(* IEC 61131-3 sources: beckhoffAutomationInterface/ST/Shark/App/Shark/Config/Machine, 12 files *)

(* ---- GVL_ChuckVacuumSystem.st ---- *)
(* CONFIG_TIER: 1-MACHINE  -- Update all values for every new machine build. *)
(* Chuck vacuum zone size thresholds for the Shark system.
   Maps wafer diameter [mm] to vacuum zone selection:
     diameter <= CHUCK_ZONE_SMALL_MAX  -> zone 1 (small)
     diameter <= CHUCK_ZONE_MEDIUM_MAX -> zone 2 (medium)
     diameter >  CHUCK_ZONE_MEDIUM_MAX -> zone 3 (large) *)
{attribute 'qualified_only'}
VAR_GLOBAL CONSTANT
    CHUCK_ZONE_SMALL_MAX  : INT := 150;   // [mm] upper bound for small-wafer zone
    CHUCK_ZONE_MEDIUM_MAX : INT := 200;   // [mm] upper bound for medium-wafer zone
END_VAR

(* ---- GVL_DIOConfig.st ---- *)
(* CONFIG_TIER: 1-MACHINE  -- Update all values for every new machine build. *)
(* Digital I/O channel counts for the Shark system.
   Values must match the extent of the corresponding E_*Identifier enums.
   Absorbs the old GVL_DigitalInputSystem and GVL_DigitalOutputSystem files. *)
{attribute 'qualified_only'}
VAR_GLOBAL CONSTANT
    // Digital I/O channel counts (must match the extent of their E_*Identifier enums)
    DI_COUNT : INT := 12;   // E_DigitalInputIdentifier  (was GVL_DigitalInputSystem.INPUT_COUNT)
    DO_COUNT : INT := 16;   // E_DigitalOutputIdentifier (was GVL_DigitalOutputSystem.OUTPUT_COUNT)

    // Outputs activated once on first boot (section 8 one-time init)
    // To add a new auto-start output: increment AUTO_START_DO_COUNT and add the identifier.
    AUTO_START_DO_COUNT   : INT := 3;
    AUTO_START_DO_OUTPUTS : ARRAY[1..3] OF INT := [
        E_DigitalOutputIdentifier.LGHT_CMR_TOP,    // Top camera light
        E_DigitalOutputIdentifier.LGHT_CMR_SIDE,   // Side camera light
        E_DigitalOutputIdentifier.CHIL_PWR         // Chiller power
    ];
END_VAR

(* ---- GVL_DoorSystem.st ---- *)
(* CONFIG_TIER: 1-MACHINE  -- Update all values for every new machine build. *)
(* Door subsystem sizing constants for the Shark system.
   DOOR_SENSOR_COUNT must match the number of proximity sensors wired
   to E_DigitalInputIdentifier door entries.
   DOOR_LOCK_COUNT must match the number of electromechanical locks
   wired to E_DigitalOutputIdentifier lock entries (FL, FR). *)
{attribute 'qualified_only'}
VAR_GLOBAL CONSTANT
    DOOR_SENSOR_COUNT : INT := 9;   // Proximity sensors total
    DOOR_LOCK_COUNT   : INT := 2;   // Electromechanical locks (FL, FR)
END_VAR

(* ---- GVL_FlowSystem.st ---- *)
(* CONFIG_TIER: 1-MACHINE  -- Update all values for every new machine build. *)
{attribute 'qualified_only'}
VAR_GLOBAL CONSTANT
    // Flow Ranges - Precursor MFC (0-25 sccm)
    MIN_FLOW_PRECURSOR_SCCM : REAL := 0.0;
    MAX_FLOW_PRECURSOR_SCCM : REAL := 25.0;

    // Flow Ranges - Reactant MFC (0-25 sccm)
    MIN_FLOW_REACTANT_SCCM  : REAL := 0.0;
    MAX_FLOW_REACTANT_SCCM  : REAL := 25.0;

    // Flow Ranges - Inert MFC (0-500 sccm)
    MIN_FLOW_INERT_SCCM     : REAL := 0.0;
    MAX_FLOW_INERT_SCCM     : REAL := 500.0;

    // System Configuration
    FLOW_ZONE_COUNT          : INT := 3;

    // Tolerance for setpoint boundary detection
    SETPOINT_TOLERANCE       : REAL := 0.01;
END_VAR

(* ---- GVL_HumiditySystem.st ---- *)
(* CONFIG_TIER: 1-MACHINE  -- Update all values for every new machine build.
   Scaling for the MDP5001_300_7E2119CA humidity channel on the Shark TH sensor pair.
   Humidity channel uses standard 0-30518 full-scale.
   Temperature channel has moved to GVL_TemperatureSystem (AMBT_TEMP_*). *)
{attribute 'qualified_only'}
VAR_GLOBAL CONSTANT
    // AMBT_HUMID: Ambient relative humidity [%RH]
    AMBT_HUMID_RAW_MIN    : LREAL := 0.0;
    AMBT_HUMID_RAW_MAX    : LREAL := 30518.0;
    AMBT_HUMID_SCALED_MIN : LREAL := 0.0;    // %RH
    AMBT_HUMID_SCALED_MAX : LREAL := 100.0;  // %RH

END_VAR

(* ---- GVL_PressureSystem.st ---- *)
(* CONFIG_TIER: 1-MACHINE  -- Update all values for every new machine build. *)
{attribute 'qualified_only'}
VAR_GLOBAL CONSTANT
    // Pressure Sensor Count (analog read-only sensors)
    SENSOR_COUNT     : INT := 4;

    // Pressure Controller Count (Bronkhorst Modbus, managed by PRG_BronkhorstPressure)
    CONTROLLER_COUNT : INT := 2;

    // Pressure Limits
    MIN_PRESSURE_BAR : REAL := 0.0;
    MAX_PRESSURE_BAR : REAL := 3.0;

    // Pressure Controller Constants (Bronkhorst Modbus needle valves)
    MIN_PRESSURE_CTRL_BAR  : REAL := 0.0;
    MAX_PRESSURE_CTRL_BAR  : REAL := 3.0;
    SETPOINT_TOLERANCE     : REAL := 0.01;
    MODBUS_FIRST_SLAVE_ADDRESS : BYTE := 1;

    // Sensor-specific raw scaling (from old FB_PressureSensorManager)
    // PSNS_A_DST: 0-30518 raw → 0.0-3.0 bar(a)
    PSNS_A_DST_RAW_MIN      : LREAL := 0.0;
    PSNS_A_DST_RAW_MAX      : LREAL := 30518.0;
    PSNS_A_DST_SCALED_MIN   : LREAL := 0.0;
    PSNS_A_DST_SCALED_MAX   : LREAL := 3.0;

    // PSNS_B_DST: 0-30518 raw → 0.0-3.0 bar(a)
    PSNS_B_DST_RAW_MIN      : LREAL := 0.0;
    PSNS_B_DST_RAW_MAX      : LREAL := 30518.0;
    PSNS_B_DST_SCALED_MIN   : LREAL := 0.0;
    PSNS_B_DST_SCALED_MAX   : LREAL := 3.0;

    // PSNS_AB_EXH: 0-30518 raw → 0.0-1.0 bar(a)
    PSNS_AB_EXH_RAW_MIN     : LREAL := 0.0;
    PSNS_AB_EXH_RAW_MAX     : LREAL := 30518.0;
    PSNS_AB_EXH_SCALED_MIN  : LREAL := 0.0;
    PSNS_AB_EXH_SCALED_MAX  : LREAL := 1.0;

    // PSNS_CHK_VAC: 3052-15259 raw → 1.01325-0.00325 bar(a) [INVERTED]
    // NOTE: Physical relationship is inverted — higher raw = lower pressure (more vacuum).
    //       FB_AnalogSensor requires ascending ranges, so we store ascending params here.
    //       Reading will be physically inverted: actual_bar = 1.0165 - sensor_reading
    PSNS_CHK_VAC_RAW_MIN    : LREAL := 3052.0;
    PSNS_CHK_VAC_RAW_MAX    : LREAL := 15259.0;
    PSNS_CHK_VAC_SCALED_MIN : LREAL := 0.00325;
    PSNS_CHK_VAC_SCALED_MAX : LREAL := 1.01325;
END_VAR

(* ---- GVL_Spectrometer.st ---- *)
(* CONFIG_TIER: 1-MACHINE  -- Update all values for every new machine build. *)
{attribute 'qualified_only'}
VAR_GLOBAL CONSTANT
    // Pixel count of the installed spectrometer detector array
    SPECTROMETER_PIXEL_COUNT : INT := 2048;
END_VAR

(* ---- GVL_System.st ---- *)
(* CONFIG_TIER: 1-MACHINE  -- Update all values for every new machine build. *)
(*
Global system state — Shark system.
From old GVL_System.st: system-wide flags and identity.
*)
{attribute 'qualified_only'}
VAR_GLOBAL
    bSystemInitialized      : BOOL := FALSE;
    bSystemHealthy          : BOOL := FALSE;
    bGlobalEmergencyStop    : BOOL := FALSE;
    bGlobalSafetyOK         : BOOL := FALSE;
    sSystemName             : STRING(80) := 'PLC_SHARK_PROJ';
    sSystemVersion          : STRING(20) := '1.2.0';
END_VAR

(* ---- GVL_TemperatureZoneConfig.st ---- *)
(* CONFIG_TIER: 1-MACHINE  -- Update all values for every new machine build. *)
(* Per-zone configuration table for the Shark temperature subsystem.
   Indexed by E_HeatZone. Each row describes ONE logical heat zone
   (composed of nChannelCount independent channel controllers).

   PID gains are NOT here: they are per-channel, in PID_GAINS (below),
   indexed by global channel index. Each channel of a zone may be tuned
   independently. *)
{attribute 'qualified_only'}
VAR_GLOBAL CONSTANT
    ZONE_CONFIG : ARRAY[1..GVL_TemperatureZones.CONTROLLABLE_ZONE_MAX] OF ST_TemperatureZoneConfig := [

        // Zone 1: HETR_HEAD - shared head heater (single channel)
        (bPopulated := TRUE,
            nChannelCount := 1,
            eAggregation := E_TempAggregation.MASTER,
            rMaxDeltaWarn := 0.0,  rMaxDeltaTrip := 0.0,
            rMinSetpoint := 20.0,  rMaxSetpoint := 150.0,
            rHeatingRampRate := 2.0,  rCoolingRampRate := 0.0),

        // Zone 2: HETR_A_STR - A-side umbilical (single channel)
        (bPopulated := TRUE,
            nChannelCount := 1,
            eAggregation := E_TempAggregation.MASTER,
            rMaxDeltaWarn := 0.0,  rMaxDeltaTrip := 0.0,
            rMinSetpoint := 20.0,  rMaxSetpoint := 140.0,
            rHeatingRampRate := 2.0,  rCoolingRampRate := 0.0),

        // Zone 3: HETR_A_CMB - A-side hot combiner / manifold (single channel)
        (bPopulated := TRUE,
            nChannelCount := 1,
            eAggregation := E_TempAggregation.MASTER,
            rMaxDeltaWarn := 0.0,  rMaxDeltaTrip := 0.0,
            rMinSetpoint := 20.0,  rMaxSetpoint := 140.0,
            rHeatingRampRate := 2.0,  rCoolingRampRate := 0.0),

        // Zone 4: HETR_A_B1 - A-side bubbler 1 (single channel)
        (bPopulated := TRUE,
            nChannelCount := 1,
            eAggregation := E_TempAggregation.MASTER,
            rMaxDeltaWarn := 0.0,  rMaxDeltaTrip := 0.0,
            rMinSetpoint := 20.0,  rMaxSetpoint := 140.0,
            rHeatingRampRate := 2.0,  rCoolingRampRate := 0.0),

        // Zone 5: HETR_A_B2 - A-side bubbler 2 (single channel)
        (bPopulated := TRUE,
            nChannelCount := 1,
            eAggregation := E_TempAggregation.MASTER,
            rMaxDeltaWarn := 0.0,  rMaxDeltaTrip := 0.0,
            rMinSetpoint := 20.0,  rMaxSetpoint := 140.0,
            rHeatingRampRate := 2.0,  rCoolingRampRate := 0.0),

        // Zone 6: HETR_A_B3 - A-side bubbler 3 (single channel)
        (bPopulated := TRUE,
            nChannelCount := 1,
            eAggregation := E_TempAggregation.MASTER,
            rMaxDeltaWarn := 0.0,  rMaxDeltaTrip := 0.0,
            rMinSetpoint := 20.0,  rMaxSetpoint := 140.0,
            rHeatingRampRate := 2.0,  rCoolingRampRate := 0.0),

        // Zone 7: HETR_B_STR - B-side umbilical (single channel)
        (bPopulated := TRUE,
            nChannelCount := 1,
            eAggregation := E_TempAggregation.MASTER,
            rMaxDeltaWarn := 0.0,  rMaxDeltaTrip := 0.0,
            rMinSetpoint := 20.0,  rMaxSetpoint := 140.0,
            rHeatingRampRate := 2.0,  rCoolingRampRate := 0.0),

        // Zone 8: HETR_B_CMB - B-side hot combiner / manifold (single channel)
        (bPopulated := TRUE,
            nChannelCount := 1,
            eAggregation := E_TempAggregation.MASTER,
            rMaxDeltaWarn := 0.0,  rMaxDeltaTrip := 0.0,
            rMinSetpoint := 20.0,  rMaxSetpoint := 140.0,
            rHeatingRampRate := 2.0,  rCoolingRampRate := 0.0),

        // Zone 9: HETR_B_B1 - B-side bubbler 1 (single channel)
        (bPopulated := TRUE,
            nChannelCount := 1,
            eAggregation := E_TempAggregation.MASTER,
            rMaxDeltaWarn := 0.0,  rMaxDeltaTrip := 0.0,
            rMinSetpoint := 20.0,  rMaxSetpoint := 140.0,
            rHeatingRampRate := 2.0,  rCoolingRampRate := 0.0),

        // Zone 10: HETR_B_B2 - B-side bubbler 2 (single channel)
        (bPopulated := TRUE,
            nChannelCount := 1,
            eAggregation := E_TempAggregation.MASTER,
            rMaxDeltaWarn := 0.0,  rMaxDeltaTrip := 0.0,
            rMinSetpoint := 20.0,  rMaxSetpoint := 140.0,
            rHeatingRampRate := 2.0,  rCoolingRampRate := 0.0),

        // Zone 11: HETR_B_B3 - B-side bubbler 3 (single channel)
        (bPopulated := TRUE,
            nChannelCount := 1,
            eAggregation := E_TempAggregation.MASTER,
            rMaxDeltaWarn := 0.0,  rMaxDeltaTrip := 0.0,
            rMinSetpoint := 20.0,  rMaxSetpoint := 140.0,
            rHeatingRampRate := 2.0,  rCoolingRampRate := 0.0),

        // Zone 12: HETR_EXH - Exhaust (2 channels: inner + outer)
        // Looser delta-trip; end segment loses heat faster than centre.
        (bPopulated := TRUE,
            nChannelCount := 2,
            eAggregation := E_TempAggregation.AVERAGE,
            rMaxDeltaWarn := 8.0,  rMaxDeltaTrip := 25.0,
            rMinSetpoint := 20.0,  rMaxSetpoint := 160.0,
            rHeatingRampRate := 2.0,  rCoolingRampRate := 0.0),

        // Zone 13: HETR_CHK - Chuck (2 channels: inner + outer)
        // Tight delta - wafer thermal coupling requires synchronised inner/outer.
        // Replaces the old FB_BeckhoffDualZoneCoord pair coordination.
        (bPopulated := TRUE,
            nChannelCount := 2,
            eAggregation := E_TempAggregation.AVERAGE,
            rMaxDeltaWarn := 3.0,  rMaxDeltaTrip := 10.0,
            rMinSetpoint := 20.0,  rMaxSetpoint := 300.0,
            rHeatingRampRate := 0.0,  rCoolingRampRate := 0.0)
    ];

    // -----------------------------------------------------------------------
    // PER-CHANNEL MAXIMUM DUTY CYCLE (heater output cap, %)
    // -----------------------------------------------------------------------
    // Hardware-imposed maximum heater duty cycle per channel (flat globalIdx
    // 1..CHANNEL_MAX, same ordering as PRG_TEMPERATURE_SENSOR / PRG_HEAT_ZONE).
    // Applied as the controller output cap (fYMax) AND clamps the autotune step,
    // so a channel can never exceed its rating even during tuning.
    // SAFETY/HARDWARE-CRITICAL: commissioning-signed values. Default 60 %.
    //
    // Channel layout (15 channels):
    //   1 HETR_HEAD   2 HETR_A_STR  3 HETR_A_CMB  4 HETR_A_B1  5 HETR_A_B2
    //   6 HETR_A_B3   7 HETR_B_STR  8 HETR_B_CMB  9 HETR_B_B1  10 HETR_B_B2
    //   11 HETR_B_B3  12..13 HETR_EXH (inner+outer)  14..15 HETR_CHK (inner+outer)
    MAX_DUTY_CYCLE : ARRAY[1..GVL_TemperatureZones.CHANNEL_MAX] OF LREAL := [
        90.0,  // 1 HETR_HEAD
        60.0,  // 2 HETR_A_STR
        60.0,  // 3 HETR_A_CMB
        60.0,  // 4 HETR_A_B1
        60.0,  // 5 HETR_A_B2
        60.0,  // 6 HETR_A_B3
        60.0,  // 7 HETR_B_STR
        60.0,  // 8 HETR_B_CMB
        60.0,  // 9 HETR_B_B1
        60.0,  // 10 HETR_B_B2
        60.0,  // 11 HETR_B_B3
        60.0,  // 12 HETR_EXH (inner)
        60.0,  // 13 HETR_EXH (outer)
        60.0,  // 14 HETR_CHK (inner)
        60.0   // 15 HETR_CHK (outer)
    ];

    // -----------------------------------------------------------------------
    // PER-CHANNEL PID GAINS (one tuned gain set per heater channel)
    // -----------------------------------------------------------------------
    // Flat per-channel PID gains (globalIdx 1..CHANNEL_MAX, same ordering as
    // PRG_TEMPERATURE_SENSOR / PRG_HEAT_ZONE). Channels within a zone are
    // physically distinct bands and may each need different gains; the Beckhoff
    // autotune produces a per-channel result, so this table is the single place
    // to record tuned gains.
    //
    // Team tuning policy: tune one channel with all channels of the zone active
    // at the same setpoint, then copy the resulting gains into that channel's
    // row. Channels seeded with their zone's previous shared gains.
    //
    // Channel layout (15 channels):
    //   1 HETR_HEAD   2 HETR_A_STR  3 HETR_A_CMB  4 HETR_A_B1  5 HETR_A_B2
    //   6 HETR_A_B3   7 HETR_B_STR  8 HETR_B_CMB  9 HETR_B_B1  10 HETR_B_B2
    //   11 HETR_B_B3  12..13 HETR_EXH (inner+outer)  14..15 HETR_CHK (inner+outer)
    PID_GAINS : ARRAY[1..GVL_TemperatureZones.CHANNEL_MAX] OF ST_HeatChannelPIDGains := [
        (rKp := 23.0, tTn := T#1m20s, tTv := T#22s, tTd := T#6s),  // 1 HETR_HEAD
        (rKp := 7.0,  tTn := T#1m50s, tTv := T#31s, tTd := T#8s),  // 2 HETR_A_STR
        (rKp := 24.0, tTn := T#1m,    tTv := T#16s, tTd := T#4s),  // 3 HETR_A_CMB
        (rKp := 9.0,  tTn := T#40s,   tTv := T#11s, tTd := T#3s),  // 4 HETR_A_B1
        (rKp := 9.0,  tTn := T#40s,   tTv := T#11s, tTd := T#3s),  // 5 HETR_A_B2
        (rKp := 9.0,  tTn := T#40s,   tTv := T#11s, tTd := T#3s),  // 6 HETR_A_B3
        (rKp := 9.5,  tTn := T#1m20s, tTv := T#22s, tTd := T#5s),  // 7 HETR_B_STR
        (rKp := 18.0, tTn := T#1m10s, tTv := T#19s, tTd := T#5s),  // 8 HETR_B_CMB
        (rKp := 9.0,  tTn := T#40s,   tTv := T#11s, tTd := T#3s),  // 9 HETR_B_B1
        (rKp := 9.0,  tTn := T#40s,   tTv := T#11s, tTd := T#3s),  // 10 HETR_B_B2
        (rKp := 9.0,  tTn := T#40s,   tTv := T#11s, tTd := T#3s),  // 11 HETR_B_B3
        (rKp := 5.0,  tTn := T#2m,    tTv := T#30s, tTd := T#8s),  // 12 HETR_EXH (inner)
        (rKp := 5.0,  tTn := T#2m,    tTv := T#30s, tTd := T#8s),  // 13 HETR_EXH (outer)
        (rKp := 12.0, tTn := T#45s,   tTv := T#12s, tTd := T#3s),  // 14 HETR_CHK (inner)
        (rKp := 12.0, tTn := T#45s,   tTv := T#12s, tTd := T#3s)   // 15 HETR_CHK (outer)
    ];

    // -----------------------------------------------------------------------
    // PER-CHANNEL DUAL-RTD DEVIATION LIMIT (°C)
    // -----------------------------------------------------------------------
    // Max allowed difference between a channel's A/B RTDs before FB_DualSensor
    // raises ERR_CTRL_DEVIATION_HIGH. Per channel because each band's RTD pair
    // sees a different physical gradient, so one global limit does not fit all.
    // Same global-index ordering as PID_GAINS / PRG_TEMPERATURE_SENSOR.
    // Single-RTD channels (CHK 14..15) run FB_DualSensor in single mode and
    // ignore this value (no pair to compare).
    //
    // Channel layout (15 channels):
    //   1 HETR_HEAD   2 HETR_A_STR  3 HETR_A_CMB  4 HETR_A_B1  5 HETR_A_B2
    //   6 HETR_A_B3   7 HETR_B_STR  8 HETR_B_CMB  9 HETR_B_B1  10 HETR_B_B2
    //   11 HETR_B_B3  12..13 HETR_EXH (inner+outer)  14..15 HETR_CHK (inner+outer)
    CHANNEL_MAX_DEVIATION : ARRAY[1..GVL_TemperatureZones.CHANNEL_MAX] OF LREAL := [
        30.0,  // 1 HETR_HEAD
        30.0,  // 2 HETR_A_STR
        30.0,  // 3 HETR_A_CMB  — raised from 15.0: physical RTD spread 15-17 °C, was nuisance-tripping at 15.0
        30.0,  // 4 HETR_A_B1
        30.0,  // 5 HETR_A_B2
        30.0,  // 6 HETR_A_B3   — raised from 15.0: physical RTD spread 15-17 °C, was nuisance-tripping at 15.0
        30.0,  // 7 HETR_B_STR
        30.0,  // 8 HETR_B_CMB
        30.0,  // 9 HETR_B_B1
        30.0,  // 10 HETR_B_B2
        30.0,  // 11 HETR_B_B3
        30.0,  // 12 HETR_EXH (inner)
        30.0,  // 13 HETR_EXH (outer)
        15.0,  // 14 HETR_CHK (inner)
        15.0   // 15 HETR_CHK (outer)
    ];
END_VAR

(* ---- GVL_TemperatureZones.st ---- *)
(* CONFIG_TIER: 1-MACHINE  -- Update all values for every new machine build. *)
(* Array bound constants for the Shark temperature subsystem.
   Heat zones:        1-13 (E_HeatZone)
   Monitor points:      1-4  (E_TemperatureMonitorZone)
   Per-zone channels: 1..GVL_HeatZone.MAX_CHANNELS (Lib constant)
   Total channels (sum of nChannelCount across zones):
     HEAD (shared)      = 1
     A-side singles     = 5 * 1 = 5
     B-side singles     = 5 * 1 = 5
     EXH (2) + CHK (2)  = 4
     Total              = 15 *)
{attribute 'qualified_only'}
VAR_GLOBAL CONSTANT
    CONTROLLABLE_ZONE_MAX : INT := 13;  // Zone count (matches highest E_HeatZone value)
    CHANNEL_MAX           : INT := 15;  // Sum of nChannelCount across all zones
    MONITOR_ZONE_COUNT    : INT := 5;   // Monitor points 1-5 (E_TemperatureMonitorZone); 1=SENS_CHAMBER, 2=SENS_STAGE_X, 3=SENS_STAGE_Y, 4=SENS_A_SIDE, 5=SENS_B_SIDE; all wired on Shark
END_VAR

(* ---- GVL_ValveSystem.st ---- *)
(* CONFIG_TIER: 1-MACHINE  -- Update all values for every new machine build. *)
{attribute 'qualified_only'}
VAR_GLOBAL CONSTANT
    // Valve counts by type
    PNEUMATIC_VALVE_COUNT  : INT := 29;  // SMC Block: valves 1-29
    SOLENOID_VALVE_COUNT   : INT := 6;   // Digital outputs: valves 30-35
    VALVE_COUNT            : INT := 35;
END_VAR

(* ---- GVL_Version.st ---- *)
(* CONFIG_TIER: 1-MACHINE  -- Update all values for every new machine build. *)
(*
Project version — Shark system.
Replaces old Global_Version.st + F_GetVersion.st.
*)
{attribute 'qualified_only'}
VAR_GLOBAL CONSTANT
    stLibVersion : ST_LibVersion := (
        iMajor   := 1,
        iMinor   := 2,
        iBuild   := 0,
        iRevision := 0,
        sVersion := '1.2.0'
    );
END_VAR
